FUNCTION_BLOCK FB_HLK (*System Heizung Lueftung Klimatisierung*)
VAR_INPUT
END_VAR
VAR_OUTPUT
END_VAR
VAR

	Tempfuehler_Rueckl_Wand_Ost_Sektor1		: FB_TF;
	Tempfuehler_Rueckl_Wand_Ost_Sektor2		: FB_TF;
	Tempfuehler_Rueckl_Wand_Ost_Sektor3		: FB_TF;
	Tempfuehler_Rueckl_Wand_West_Sektor1	: FB_TF;
	Tempfuehler_Rueckl_Wand_West_Sektor2	: FB_TF;
	Tempfuehler_Rueckl_Wand_West_Sektor3	: FB_TF;
	Tempfuehler_Rueckl_Decke_Ost_Sektor1	: FB_TF;
	Tempfuehler_Rueckl_Decke_Ost_Sektor2	: FB_TF;
	Tempfuehler_Rueckl_Decke_Ost_Sektor3	: FB_TF;
	Tempfuehler_Rueckl_Decke_West_Sektor1	: FB_TF;
	Tempfuehler_Rueckl_Decke_West_Sektor2	: FB_TF;
	Tempfuehler_Rueckl_Decke_West_Sektor3	: FB_TF;
	Tempfuehler_Rueckl_Aussen_Ost			: FB_TF;
	Tempfuehler_Rueckl_Aussen_West			: FB_TF;
	Temp_Aussen_WS        					: FB_TF;

	System_Fussbodentemperierung_425		: FB_System_FBT_425;
	System_Wanddeckentemperierung_500		: FB_System_WDT_500;
	System_Lueftungsanlage_955				: FB_System_LA_955;
	System_StatischeHeizung_350				: FB_System_SHZ_350;

	Fenster									: FB_System_Fenster;
	DS_500_Wand_Innen						: FB_DS;
	DS_600_Wand_Aussen						: FB_DS;
END_VAR

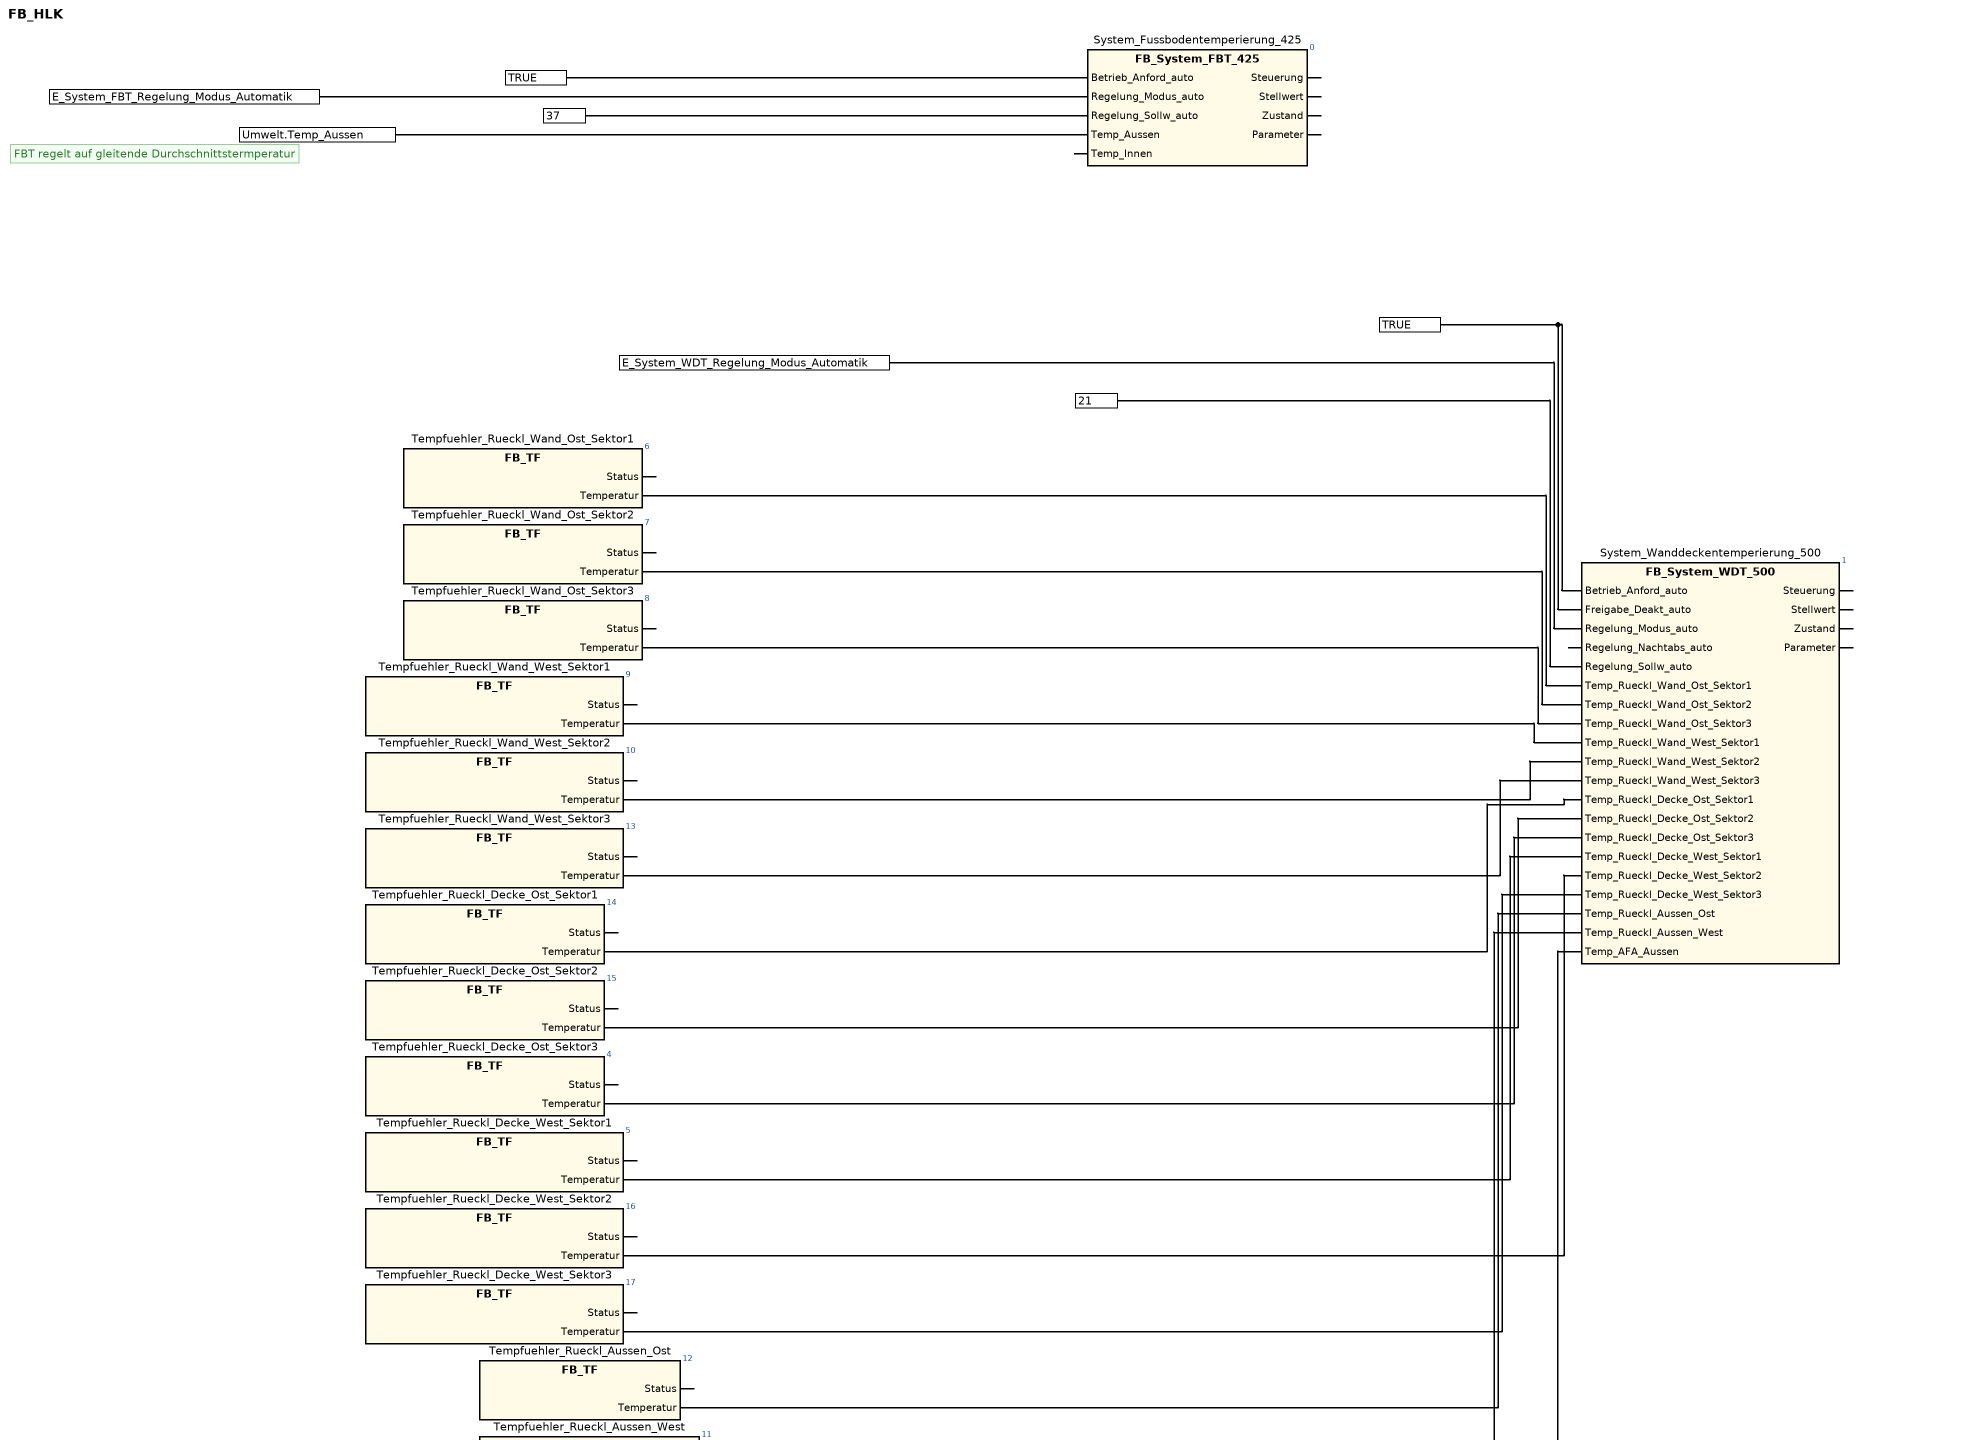
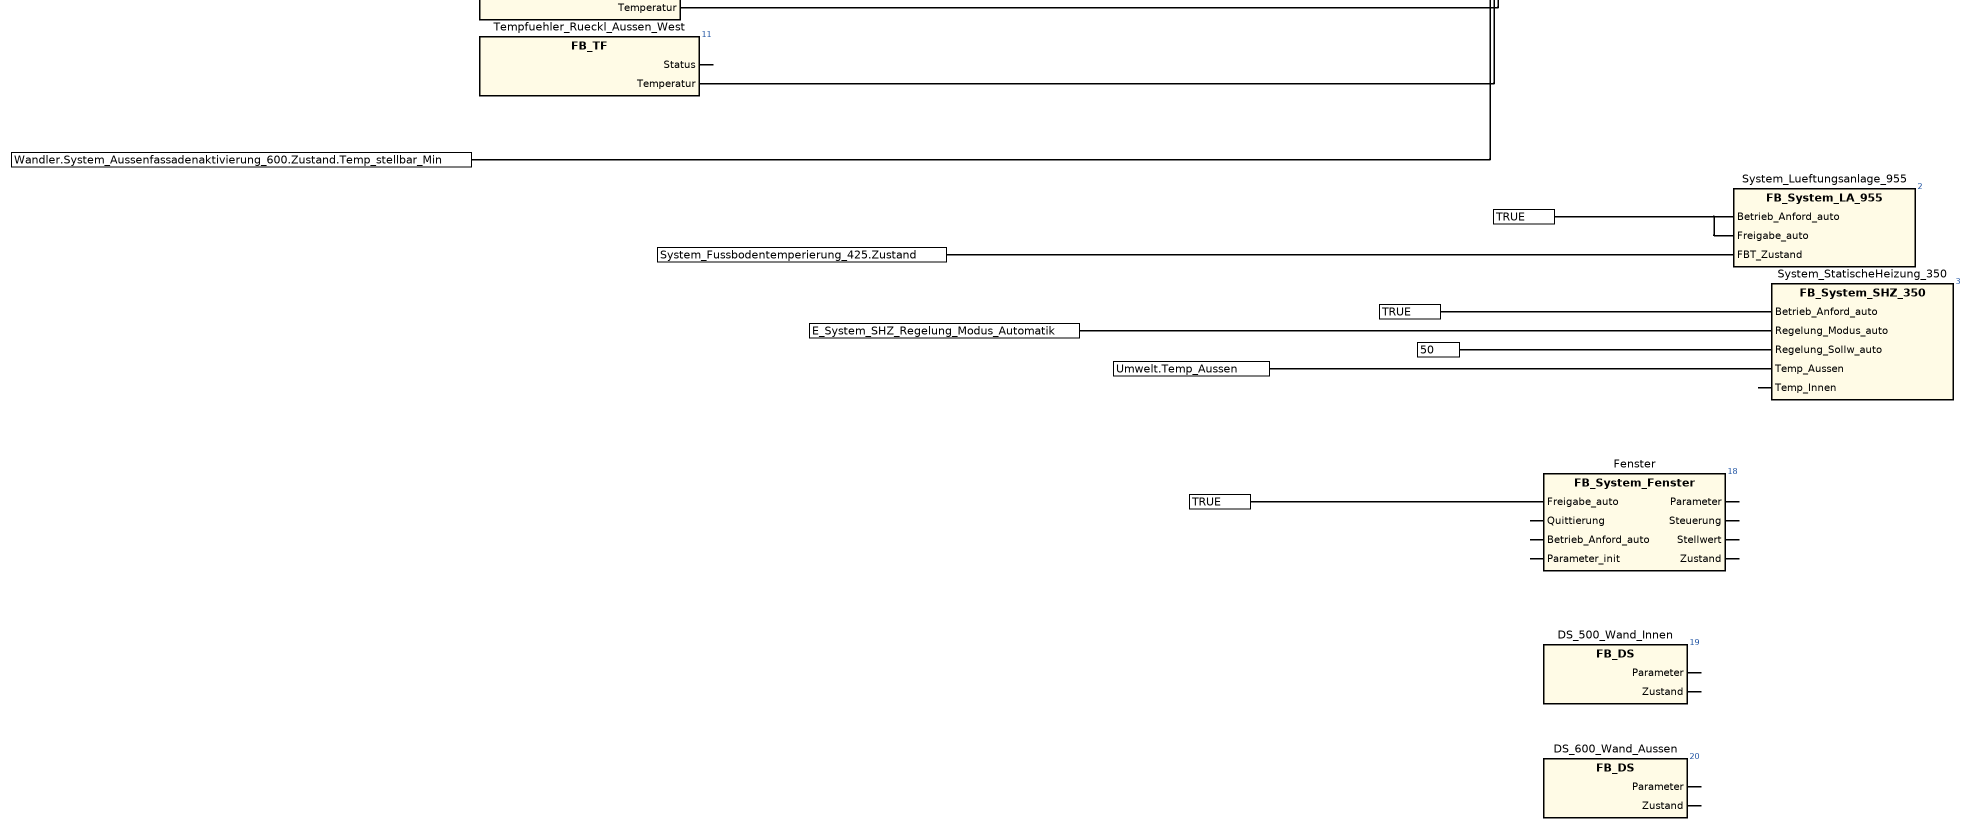
System_Fussbodentemperierung_425(
    Betrieb_Anford_auto := TRUE,
    Regelung_Modus_auto := E_System_FBT_Regelung_Modus_Automatik,
    Regelung_Sollw_auto := 37,
    Temp_Aussen := Umwelt.Temp_Aussen); // FB_System_FBT_425
System_Wanddeckentemperierung_500(
    Betrieb_Anford_auto := TRUE,
    Freigabe_Deakt_auto := TRUE,
    Regelung_Modus_auto := E_System_WDT_Regelung_Modus_Automatik,
    Regelung_Sollw_auto := 21,
    Temp_Rueckl_Wand_Ost_Sektor1 := Tempfuehler_Rueckl_Wand_Ost_Sektor1.Temperatur,
    Temp_Rueckl_Wand_Ost_Sektor2 := Tempfuehler_Rueckl_Wand_Ost_Sektor2.Temperatur,
    Temp_Rueckl_Wand_Ost_Sektor3 := Tempfuehler_Rueckl_Wand_Ost_Sektor3.Temperatur,
    Temp_Rueckl_Wand_West_Sektor1 := Tempfuehler_Rueckl_Wand_West_Sektor1.Temperatur,
    Temp_Rueckl_Wand_West_Sektor2 := Tempfuehler_Rueckl_Wand_West_Sektor2.Temperatur,
    Temp_Rueckl_Wand_West_Sektor3 := Tempfuehler_Rueckl_Wand_West_Sektor3.Temperatur,
    Temp_Rueckl_Decke_Ost_Sektor1 := Tempfuehler_Rueckl_Decke_Ost_Sektor1.Temperatur,
    Temp_Rueckl_Decke_Ost_Sektor2 := Tempfuehler_Rueckl_Decke_Ost_Sektor2.Temperatur,
    Temp_Rueckl_Decke_Ost_Sektor3 := Tempfuehler_Rueckl_Decke_Ost_Sektor3.Temperatur,
    Temp_Rueckl_Decke_West_Sektor1 := Tempfuehler_Rueckl_Decke_West_Sektor1.Temperatur,
    Temp_Rueckl_Decke_West_Sektor2 := Tempfuehler_Rueckl_Decke_West_Sektor2.Temperatur,
    Temp_Rueckl_Decke_West_Sektor3 := Tempfuehler_Rueckl_Decke_West_Sektor3.Temperatur,
    Temp_Rueckl_Aussen_Ost := Tempfuehler_Rueckl_Aussen_Ost.Temperatur,
    Temp_Rueckl_Aussen_West := Tempfuehler_Rueckl_Aussen_West.Temperatur,
    Temp_AFA_Aussen := Wandler.System_Aussenfassadenaktivierung_600.Zustand.Temp_stellbar_Min); // FB_System_WDT_500
System_Lueftungsanlage_955(
    Betrieb_Anford_auto := TRUE,
    Freigabe_auto := TRUE,
    FBT_Zustand := System_Fussbodentemperierung_425.Zustand); // FB_System_LA_955
System_StatischeHeizung_350(
    Betrieb_Anford_auto := TRUE,
    Regelung_Modus_auto := E_System_SHZ_Regelung_Modus_Automatik,
    Regelung_Sollw_auto := 50,
    Temp_Aussen := Umwelt.Temp_Aussen); // FB_System_SHZ_350
Tempfuehler_Rueckl_Decke_Ost_Sektor3(); // FB_TF
Tempfuehler_Rueckl_Decke_West_Sektor1(); // FB_TF
// FBT regelt auf gleitende Durchschnittstermperatur
Tempfuehler_Rueckl_Wand_Ost_Sektor1(); // FB_TF
Tempfuehler_Rueckl_Wand_Ost_Sektor2(); // FB_TF
Tempfuehler_Rueckl_Wand_Ost_Sektor3(); // FB_TF
Tempfuehler_Rueckl_Wand_West_Sektor1(); // FB_TF
Tempfuehler_Rueckl_Wand_West_Sektor2(); // FB_TF
Tempfuehler_Rueckl_Aussen_West(); // FB_TF
Tempfuehler_Rueckl_Aussen_Ost(); // FB_TF
Tempfuehler_Rueckl_Wand_West_Sektor3(); // FB_TF
Tempfuehler_Rueckl_Decke_Ost_Sektor1(); // FB_TF
Tempfuehler_Rueckl_Decke_Ost_Sektor2(); // FB_TF
Tempfuehler_Rueckl_Decke_West_Sektor2(); // FB_TF
Tempfuehler_Rueckl_Decke_West_Sektor3(); // FB_TF
Fenster(Freigabe_auto := TRUE); // FB_System_Fenster
DS_500_Wand_Innen(); // FB_DS
DS_600_Wand_Aussen(); // FB_DS

END_FUNCTION_BLOCK

(* stored: Version 1.1.0.1, ProductVersion 3.1.4024.9
   POU FB_HLK: Id {c4b9faac-6980-478a-8e47-a7f352351a65}, SpecialFunc None *)
